{attribute 'qualified_only'}
{attribute 'strict'}
TYPE eMode :
(
	Manual := 0,
	Automatic := 1
);
END_TYPE

(* stored: Version 1.1.0.1, ProductVersion 3.1.4026.18
   DUT eMode: Id {a1b2c3d4-3333-3333-3333-333333333333} *)
